(* CODESYS project CtaSysFU_1.0.0.0.library
   Description: SYS FU Library der CTA
   Version: 1.0.0.0
   Title: CtaSysFU
   Author: SIS
   DocFormat: reStructuredText
   LanguageModelAttribute: qualified-access-only
   Placeholder: CtaSysFU
   DefaultNamespace: CtaSysFU
   CompiledLibraryCompatibilityVersion: CODESYS V3.5 SP16 Patch 3
   Company: CTA

Project tree, tasks and I/O mapping:
  libraries: Visu Utils, 4.5.0.0 (System); CtaAppBmk, 1.0.0.0 (CTA); CtaAppReport, 1.0.0.2 (CTA); VisuSymbols, 4.5.0.0 (System); CtaVisSymbols, 1.0.0.0 (CTA); CtaAppModbusSpezifikation, 1.0.0.0 (CTA)
  40 Visualizations/
    visualisation VIS_FU_BASE
    visualisation VIS_FU_BASE_ITF
    visualisation VIS_FU_BASE_QUERRY
  00000000-0000-0000-0000-000000000000|D:\CoDeSys\LibrariesV3\trunk\Intern\CAA\CAA Template\3.4.0.0 draft\Placeholder.xml
  00000000-0000-0000-0000-000000000000|D:\CoDeSys\LibrariesV3\trunk\Intern\CAA\CAA Template\3.2.0.3 draft\Prefix.pdf
  00000000-0000-0000-0000-000000000000|D:\CoDeSys\LibrariesV3\trunk\Intern\CAA\CAA Template\3.5.2.0 draft\Placeholder.xml
  20 Structs/
  50 Images/
  10 Documenation/
    global variables VersionHistory
    global variables readMe
  21 Interface/
    interface ITF_FU_BASE: proEnable, proAcknowledge, proAcknowledge_Hz, proAmpere, proBUS_OK, proError, proFU_TYPE, proReady, proRelease, proRelease_Hz, proVISU_DIA_NAME, proVolt, proQuitt, prokWatt, proTemperatur, proITF_ReportManager, proHandLokal, proModbusStateWord
  11 Library Parameter/
  12 Konstanten/
  60 Textlisten/
    text list Error
    text list Info
    text list Warnung
  13 Globale Variablen/
  text list GlobalTextList
  5ce3da45-db07-42e7-a21c-a00fff4ed8f6|C:\Users\sis\Downloads\dip-switch.svg
  5ce3da45-db07-42e7-a21c-a00fff4ed8f6|C:\Users\sis\Downloads\lightning-bolt-circle.svg
  30 Program Organization Units/
    function block FB_FU_BASE [ST]: proAcknowledge, proAcknowledge_Hz, proAmpere, proBUS_OK, proError, proFU_TYPE, proReady, proRelease, proRelease_Hz, proVISU_DIA_NAME, proVolt, proEnable, proQuitt, prokWatt, proTemperatur, proITF_ReportManager, proHandLokal, proModbusStateWord
  5ce3da45-db07-42e7-a21c-a00fff4ed8f6|C:\Users\sis\Downloads\sine-wave.svg
  5ce3da45-db07-42e7-a21c-a00fff4ed8f6|C:\Users\sis\Downloads\eye.svg
  5ce3da45-db07-42e7-a21c-a00fff4ed8f6|C:\Users\sis\Downloads\lan.svg
*)

// 10 Documenation/VersionHistory
(* 

.. image:: ../../Images/CTA_Logo.jpg
   :align: right
   :width: 15% 

**Vorlage**   


============ =========== =========== ============================================
**Date**     **Version** **Author**  **Change**
------------ ----------- ----------- --------------------------------------------
04.03.2021   0.0.0.0     SIS         Vorlage erstellt

============ =========== =========== ============================================


*)
VAR_GLOBAL
    stInfo : STRING:= '0.0.0.0, Vorlage, CTA';
END_VAR

// 10 Documenation/readMe
(*

**ReadMe**
 
|	**Empfehlung**
|
|	Dokumentrieren Sie die Library für eine nachhaltige Entwicklung
|     
| *Beispiel*
| 
| Dies ist die Vorlage Library der CTA. Erstellen Sie ihre Library anhand dieser Vorlage.
*)

VAR_GLOBAL
    xReadMeDone              :   BOOL;
END_VAR

// 30 Program Organization Units/FB_FU_BASE
FUNCTION_BLOCK FB_FU_BASE EXTENDS CtaAppBmk.fbBMK IMPLEMENTS ITF_FU_BASE
VAR
	xEnable				:	BOOL;
	xQuitt				:	BOOL;
    xReady          	:   BOOL;
    xRelease        	:   BOOL;
    rRelease_Hz     	:   REAL;
    xAcknowledge    	:   BOOL;
    rAcknowledge_Hz 	:   REAL;
    xError          	:   BOOL;  
    rAmpere         	:   REAL;
    rVolt           	:   REAL;
	rkWatt				:	REAL;  
	rTemperatur			:	REAL;
    xBusOK          	:   BOOL;
	xHandLockal			:	BOOL;
	ITF_REPORTMANAGER 	: 	CtaAppReport.ITF_REPORTMANAGER;
	ayMbStateWord       :   ARRAY[0..3] OF WORD;
	stVisuDiaName		:	STRING;
END_VAR

PROPERTY proAcknowledge : BOOL
GET
proAcknowledge := xAcknowledge;
END_GET
SET
xAcknowledge := proAcknowledge;
END_SET
END_PROPERTY

PROPERTY proAcknowledge_Hz : REAL
GET
proAcknowledge_Hz := rAcknowledge_Hz;
END_GET
SET
rAcknowledge_Hz := proAcknowledge_Hz;
END_SET
END_PROPERTY

PROPERTY proAmpere : REAL
GET
proAmpere := rAmpere;
END_GET
SET
rAmpere := proAmpere;
END_SET
END_PROPERTY

PROPERTY proBUS_OK : BOOL
GET
proBUS_OK := xBusOK;
END_GET
END_PROPERTY

PROPERTY proError : BOOL
GET
proError := xError;
END_GET
SET
xError := proError;
END_SET
END_PROPERTY

PROPERTY proFU_TYPE : STRING(20)
GET
proFU_TYPE := 'FB_FU_BASE ';
END_GET
END_PROPERTY

PROPERTY proReady : BOOL
GET
proReady := xReady;
END_GET
SET
xReady := proReady;
END_SET
END_PROPERTY

PROPERTY proRelease : BOOL
GET
proRelease := xRelease;
END_GET
SET
xRelease := proRelease;
END_SET
END_PROPERTY

PROPERTY proRelease_Hz : REAL
GET
proRelease_Hz := rRelease_Hz;
END_GET
SET
rRelease_Hz := proRelease_Hz;
END_SET
END_PROPERTY

PROPERTY proVISU_DIA_NAME : STRING
GET
proVISU_DIA_NAME := stVisuDiaName;
END_GET
END_PROPERTY

PROPERTY proVolt : REAL
GET
proVolt := rVolt;
END_GET
SET
rVolt := proVolt;
END_SET
END_PROPERTY

PROPERTY proEnable : BOOL
SET
xEnable := proEnable;
END_SET
GET
proEnable := xEnable;
END_GET
END_PROPERTY

PROPERTY proQuitt : BOOL
SET
END_SET
GET
END_GET
END_PROPERTY

PROPERTY prokWatt : REAL
SET
rkWatt := prokWatt;
END_SET
GET
prokWatt := rkWatt;
END_GET
END_PROPERTY

PROPERTY proTemperatur : REAL
SET
rTemperatur := proTemperatur;
END_SET
GET
proTemperatur := rTemperatur;
END_GET
END_PROPERTY

PROPERTY proITF_ReportManager : CtaAppReport.ITF_REPORTMANAGER;
SET
ITF_REPORTMANAGER := proITF_ReportManager;
END_SET
GET
proITF_ReportManager := ITF_REPORTMANAGER;
END_GET
END_PROPERTY

PROPERTY proHandLokal : BOOL
GET
proHandLokal := xHandLockal;
END_GET
END_PROPERTY

{warning disable C0410}
PROPERTY proModbusStateWord : REFERENCE TO ARRAY[0..3] OF WORD
{warning restore C0410}
GET
(* State Word 0 Digital Info*)
ayMbStateWord[0].00     := xRelease;
ayMbStateWord[0].01     := xAcknowledge;
ayMbStateWord[0].02     := xReady;
ayMbStateWord[0].03     := xBusOK;
ayMbStateWord[0].04     := FALSE;
ayMbStateWord[0].05     := FALSE;
ayMbStateWord[0].06     := FALSE;
ayMbStateWord[0].07     := FALSE;
ayMbStateWord[0].08     := FALSE;
ayMbStateWord[0].09     := FALSE;
ayMbStateWord[0].10     := FALSE;
ayMbStateWord[0].11     := FALSE;
ayMbStateWord[0].12     := FALSE;
ayMbStateWord[0].13     := FALSE;
ayMbStateWord[0].14     := FALSE;
ayMbStateWord[0].15     := xError;
(* VOLT *)
ayMbStateWord[1]		:= TO_WORD(rVolt * 10);
ayMbStateWord[2]		:= TO_WORD(rAmpere * 10);
ayMbStateWord[3]		:= TO_WORD(rAcknowledge_Hz * 10);

proModbusStateWord REF= ayMbStateWord;
END_GET
END_PROPERTY

END_FUNCTION_BLOCK

// 21 Interface/ITF_FU_BASE
INTERFACE ITF_FU_BASE EXTENDS CTAAppBmk.ITF_BMK , CtaAppModbusSpezifikation.ITF_MODBUS_SPEZIFIKATION

PROPERTY proEnable : BOOL
SET
END_SET
GET
END_GET
END_PROPERTY

PROPERTY proAcknowledge : BOOL
GET
END_GET
SET
END_SET
END_PROPERTY

PROPERTY proAcknowledge_Hz : REAL
GET
END_GET
SET
END_SET
END_PROPERTY

PROPERTY proAmpere : REAL
GET
END_GET
SET
END_SET
END_PROPERTY

PROPERTY proBUS_OK : BOOL
GET
END_GET
END_PROPERTY

PROPERTY proError : BOOL
GET
END_GET
SET
END_SET
END_PROPERTY

PROPERTY proFU_TYPE : STRING[20]
GET
END_GET
END_PROPERTY

PROPERTY proReady : BOOL
GET
END_GET
SET
END_SET
END_PROPERTY

PROPERTY proRelease : BOOL
GET
END_GET
SET
END_SET
END_PROPERTY

PROPERTY proRelease_Hz : REAL
GET
END_GET
SET
END_SET
END_PROPERTY

PROPERTY proVISU_DIA_NAME : STRING
GET
END_GET
END_PROPERTY

PROPERTY proVolt : REAL
GET
END_GET
SET
END_SET
END_PROPERTY

PROPERTY proQuitt : BOOL
SET
END_SET
GET
END_GET
END_PROPERTY

PROPERTY prokWatt : REAL
SET
END_SET
GET
END_GET
END_PROPERTY

PROPERTY proTemperatur : REAL
SET
END_SET
GET
END_GET
END_PROPERTY

PROPERTY proITF_ReportManager : CtaAppReport.ITF_REPORTMANAGER;
SET
END_SET
GET
END_GET
END_PROPERTY

PROPERTY proHandLokal : BOOL
GET
END_GET
END_PROPERTY

{warning disable C0410}
PROPERTY proModbusStateWord : REFERENCE TO ARRAY[0..3] OF WORD
{warning restore C0410}
GET
END_GET
END_PROPERTY

END_INTERFACE

// 40 Visualizations/VIS_FU_BASE
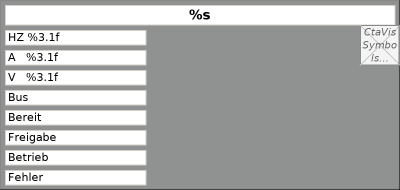
VISUALIZATION VIS_FU_BASE  // 400x190
VAR_INPUT
	ITF_FU_BASEIn   :   ITF_FU_BASE;
END_VAR
    Frame (0,0 400x190), invisible if: NOT __QUERYINTERFACE(ITF_FU_BASEIn,ITF_FU_BASEIn)
        shows VIS_FU_BASE_QUERRY(ITF_FU_BASEIn := ITF_FU_BASEIn)
END_VISUALIZATION

// 40 Visualizations/VIS_FU_BASE_ITF
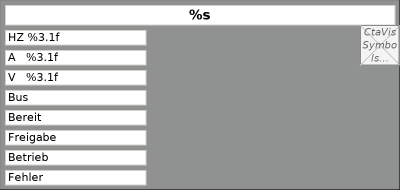
VISUALIZATION VIS_FU_BASE_ITF  // 400x190
VAR_INPUT
	ITF_FU_BASEIn   :   ITF_FU_BASE;
END_VAR
VAR
    fbDialog    	:   VU.FbOpenDialogExtended;
END_VAR
    Rectangle (0,0 400x190)
    Textfield (5,5 390x20), "%s", text variable: ITF_FU_BASEIn.proFU_TYPE
    Image (360,25 40x40), invisible if: ITF_FU_BASEIn.proVISU_DIA_NAME = '', input disabled if: ITF_FU_BASEIn.proVISU_DIA_NAME = '', image: CtaVisSymbols.ImagePool.gear
        OnMouseClick: execute {
            fbDialog(itfClientFilter            := VU.Globals.CurrentClient,
                     xExecute                   := FALSE,
                     sDialogName                := ITF_FU_BASEIn.proVISU_DIA_NAME,
                     pbyDialogInterfaceData     := ADR(ITF_FU_BASEIn),
                     udiDialogInterfaceDataSize := SIZEOF(ITF_FU_BASEIn));
            fbDialog(itfClientFilter            := VU.Globals.CurrentClient,
                     xExecute                   := TRUE,
                     sDialogName                := ITF_FU_BASEIn.proVISU_DIA_NAME,
                     pbyDialogInterfaceData     := ADR(ITF_FU_BASEIn),
                     udiDialogInterfaceDataSize := SIZEOF(ITF_FU_BASEIn));
        }
    Textfield (5,30 141x15), "HZ %3.1f", text variable: ITF_FU_BASEIn.proAcknowledge_Hz
    Textfield (5,50 141x15), "A %3.1f", text variable: ITF_FU_BASEIn.proAmpere
    Textfield (5,70 141x15), "V %3.1f", text variable: ITF_FU_BASEIn.proVolt
    Textfield (5,90 141x15), "Bus", colour toggle: ITF_FU_BASEIn.proBUS_OK
    Textfield (5,130 141x15), "Freigabe", colour toggle: ITF_FU_BASEIn.proRelease
    Textfield (5,110 141x15), "Bereit", colour toggle: ITF_FU_BASEIn.proReady
    Textfield (5,150 141x15), "Betrieb", colour toggle: ITF_FU_BASEIn.proAcknowledge
    Textfield (5,170 141x15), "Fehler", colour toggle: ITF_FU_BASEIn.proError
END_VISUALIZATION

// 40 Visualizations/VIS_FU_BASE_QUERRY
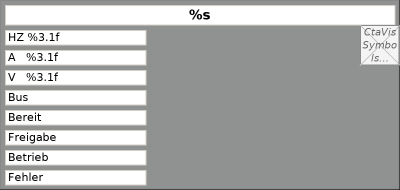
VISUALIZATION VIS_FU_BASE_QUERRY  // 400x190
VAR_INPUT
	ITF_FU_BASEIn   :   ITF_FU_BASE;
END_VAR
    Frame (0,0 400x190), invisible if: NOT ITF_FU_BASEIn.proEnable
        shows VIS_FU_BASE_ITF(ITF_FU_BASEIn := ITF_FU_BASEIn)
END_VISUALIZATION

(* text list Error (id | default | de | en | fr | it)
  0 | keine Meldung Anstehend | Keine Meldung Anstehend | No message pending | Aucun message en attente | Nessun messaggio in sospeso
  1 | keine Betriebsrückmeldung | Keine Betriebsrückmeldung | No operational feedback | Aucune rétroaction opérationnelle | Nessun feedback operativo
  2 | Alarmkontakt Anstehend | Alarmkontakt Anstehend | Error contact pending | Contact d'alarme en attente | Contatto di allarme in sospeso
  3 | Leitungsschutzschalter ausfall | Leitungsschutzschalter ausfall | Circuit breaker failure | Défaillance du disjoncteur | Guasto dell'interruttore
  4 | Motorschutzschalter ausfall | Motorschutzschalter ausfall | Motor protection switch failure | Défaillance de l'interrupteur de protection du moteur | Guasto al salvamotore
  5 | Konfigurationsfehler speichern fehlgeschlagen reboot | Konfigurationsfehler speichern fehlgeschlagen reboot | Failed to save configuration error reboot | Impossible d'enregistrer l'erreur de configuration reboot | Impossibile salvare l'errore di configurazione reboot
   |  |  |  |  |  *)

(* text list Info (id | default | de | en | fr | it)
  0 | keine Meldung Anstehend | keine Meldung Anstehend | no message pending | aucun message en attente | nessun messaggio in sospeso
   |  |  |  |  |  *)

(* text list Warnung (id | default | de | en | fr | it)
  0 | Keine Meldung Anstehend | Keine Meldung Anstehend | No message pending | Aucun message en attente | Nessun messaggio in sospeso
  4 | Wahlschalter Hand, Ein | Wahlschalter Hand, Ein | Selector switch hand on | Commutateur de sélection a main, Allumé | Selettore a mano, acceso
  3 | Wahlschalter Hand, Aus | Wahlschalter Hand, Aus | Selector switch hand off | Commutateur de sélection a main, Éteint | Selettore a mano, spento
  2 | Revisionsschalter Ausgeschalten | Revisionsschalter Ausgeschalten | Revision switch off | Commutateur révision Désactiver | Interruttore di revisione disattivato
  1 | Sicherheits Stopp | Sicherheits Stopp | Safety stop | Arrêt de sécurité | Sosta di sicurezza
  5 | Handmodul aktiv | Handmodul aktiv | Hand module active | Module manuel actif | Modulo manuale attivo
   |  |  |  |  |  *)
